PROGRAM LDPOU
VAR
	// Start Button
	btnStart: BOOL;
	// Stop Button
	btnStop: BOOL;
	// Motor Starter Coil
	Coil: BOOL;
END_VAR

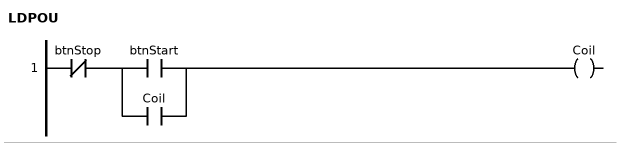
// NETWORK 1
Coil := NOT btnStop AND (btnStart OR Coil);

END_PROGRAM

(* stored: Version 1.1.0.1, ProductVersion 3.1.4024.15
   POU LDPOU: Id {fec13054-6c49-4035-8661-05acdcacbae7}, SpecialFunc None *)
